# EPICS autosave request: dxp/tags/R2-4/iocBoot/iocSaturn/auto_settings.req
file "mca_settings.req",                P=dxpSaturn:, M=mca1
file "dxp_settings.req",                P=dxpSaturn:, R=dxp1
